PROGRAM MAIN
VAR
	Machine : MachineModule := (Name := 'Machine');	
END_VAR

Machine.CyclicLogic();

END_PROGRAM

(* stored: Version 1.1.0.1, ProductVersion 3.1.4024.12
   POU MAIN: Id {c371776a-441b-42e0-8bb5-744f0ec82fd5}, SpecialFunc None *)
